INTERFACE ITF_BaseComponent_HMI_Connector_Command

END_INTERFACE

(* stored: Version 1.1.0.1
   Itf ITF_BaseComponent_HMI_Connector_Command: Id {2b2ab637-b14f-0ee4-2559-e4337058232e} *)
